INTERFACE I_Object EXTENDS __SYSTEM.IQueryInterface

END_INTERFACE

(* stored: Version 1.1.0.1
   Itf I_Object: Id {bc419bc7-e982-01ff-324b-3fdbe45e59c1} *)
